Fanuc KAREL source: kd00013.KL

-- PROVISIONAL review KL for V770-1; original PC SHA256 a6c1093a0b39a0241597ab2cd1e4c74a5ba8d05b7a6e8e51d40de0f66368f742
-- Incomplete behavior may be omitted. Consult companion uncertainty JSON. Do not deploy.
PROGRAM KD00013
%NOLOCKGROUP
VAR
  I : INTEGER
  J : INTEGER
  B : BOOLEAN
  R : REAL
  S : STRING[80]
BEGIN
  -- UNRESOLVED_PC offsets 5-13; opcodes 2E,9D,1A
  -- UNRESOLVED_PC offsets 18-22; opcodes 7F
END KD00013
